TYPE "PLCtoMES_SubCheckIn"
VERSION : 0.1
   STRUCT
      "P-SubPartID" : String[48];
      "P-SubPartReq" : Bool;
      Reserve : Array[1..247] of Byte;
   END_STRUCT;

END_TYPE

